RoboDK station: AROB_S4_A4.rdk

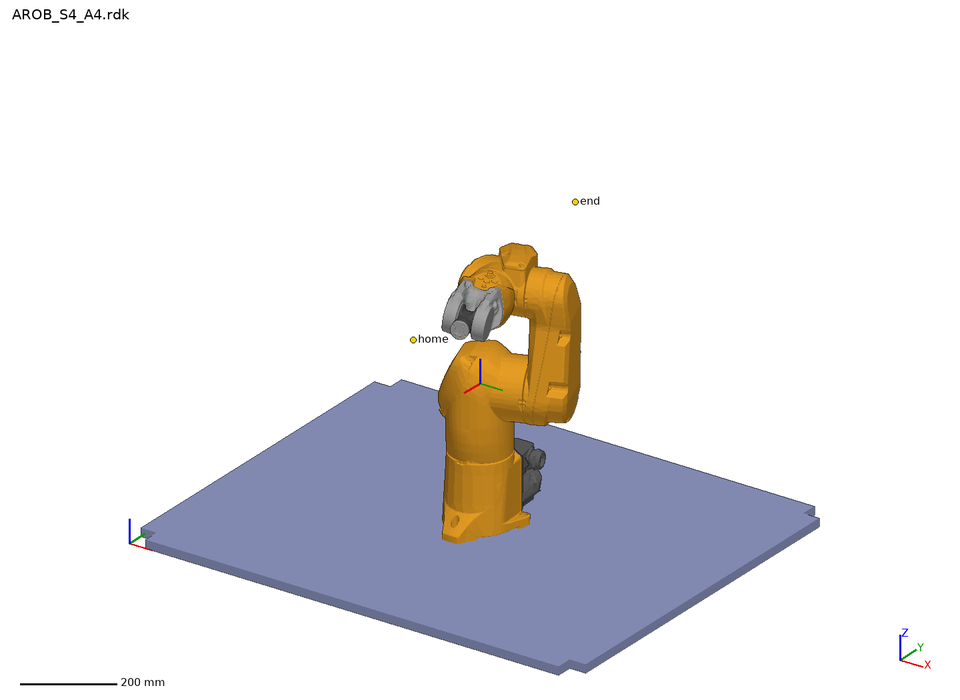
[picture v0: the station drawn from its stored meshes, robots at their saved joint values, targets as dots, program paths as lines]
Station AROB_S4_A5 (saved by RoboDK 5.6.9). Poses are relative to the parent item; angles as X-Y-Z fixed-axis rotations.
  - frame world at (0, 0, 0) mm
    - frame Staubli TX2-40 Base at (560, 460, 340) mm, rotated rx 0 ry 0 rz -90 deg
      - robot Staubli TX2-40: 6 axes, payload 2 kg, reach 515 mm, repeatability 0.02 mm, weight 29 kg
          modified DH rows (alpha deg, a mm, theta deg, d mm): 0, 0, 0, 320; -90, 0, -90, 35; 0, 225, -90, 0; -90, 0, 0, 225; 90, 0, 0, 0; -90, 0, 180, 65
          base shift (0, 0, -320) mm
          joint limits [-180, -125, -138, -270, -120, -270] to [180, 125, 138, 270, 133.5, 270]; home [0, 0, 90, 0, 0, 0]; saved at [19.667, 0, 81.667, -8.333, 5.5, 15.833]
    - object Arbeitsflaeche_geteilt at (0, 0, 0) mm, size 1120 x 920 x 20 mm, geometry from Arbeitsflaeche_geteilt.iges
    - object Arbeitsflaeche_komplett at (0, 0, 0) mm, size 1120 x 920 x 20 mm, geometry from Arbeitsflaeche_komplett.IGS
    - object Zelle at (0, 0, 0) mm, rotated rx 90 ry 0 rz -90 deg, size 1120 x 1947.8 x 1200 mm, geometry from Zelle.stp
    - target home (joint target) at (595, 170, 565) mm, rotated rx 0 ry 90 rz -90 deg; joints [0, 0, 90, 0, 0, 0] of Staubli TX2-40
    - target end (joint target) at (730.33, 559.49, 764.49) mm, rotated rx 62.55 ry 25.09 rz 78.25 deg; joints [118, 0, 40, -50, 33, 95] of Staubli TX2-40
  - Python program Prog_viaTarget (listed below)
  - Python program Prog_Direct (listed below)

--- Python program Prog_viaTarget ---
# Type help("robodk.robolink") or help("robodk.robomath") for more information
# Press F5 to run the script
# Documentation: https://robodk.com/doc/en/RoboDK-API.html
# Reference:     https://robodk.com/doc/en/PythonAPI/robodk.html
# Note: It is not required to keep a copy of this file, your Python script is saved with your RDK project
import robodk.robolink as rl    # Robot link toolbox
import time

# Link to RoboDK
RDK = rl.Robolink()

robot = RDK.Item('Staubli TX2-40')

world = RDK.Item('world')
home = RDK.Item('home')
target1 = RDK.Item('Target 1')
target2 = RDK.Item('Target 2')
target3 = RDK.Item('Target 3')
target4 = RDK.Item('Target 4')
target5 = RDK.Item('Target 5')
end = RDK.Item('end')

print('start')

robot.setAccelerationJoints(150)
robot.setSpeedJoints(75)

robot.MoveJ(home)
robot.MoveJ(target1)
robot.MoveJ(target2)
robot.MoveJ(target3)
robot.MoveJ(target4)
robot.MoveJ(target5)
robot.MoveJ(end)
time.sleep(0.1)
robot.MoveJ(target5)
robot.MoveJ(target4)
robot.MoveJ(target3)
robot.MoveJ(target2)
robot.MoveJ(target1)
robot.MoveJ(home)
print('end')

--- Python program Prog_Direct ---
# Type help("robodk.robolink") or help("robodk.robomath") for more information
# Press F5 to run the script
# Documentation: https://robodk.com/doc/en/RoboDK-API.html
# Reference:     https://robodk.com/doc/en/PythonAPI/robodk.html
# Note: It is not required to keep a copy of this file, your Python script is saved with your RDK project
import robodk.robolink as rl    # Robot link toolbox
import time
import numpy as np

# Link to RoboDK
RDK = rl.Robolink()

robot = RDK.Item('Staubli TX2-40')
world = RDK.Item('world')
home = RDK.Item('home')
target1 = RDK.Item('Target 1')
target2 = RDK.Item('Target 2')
target3 = RDK.Item('Target 3')
target4 = RDK.Item('Target 4')
target5 = RDK.Item('Target 5')
end = RDK.Item('end')

print('start')

robot.setAccelerationJoints(150)
robot.setSpeedJoints(75)

robot.MoveJ(home)
robot.MoveJ(end)

time.sleep(0.1)

robot.MoveJ(home)
print('end')
